// TIA Portal V18 export
// export: Created 2026-03-12T16:04:35.2784155Z, ExportSetting WithDefaults, DisplayName Totally Integrated Automation Portal, DisplayVersion V18 Update 5, DisplayName TIA Portal Openness, DisplayVersion V18 Update 5, DisplayName TIA Portal Version Control Interface, DisplayVersion V18, DisplayName SINAMICS Startdrive Advanced, DisplayVersion V18, DisplayName SINAMICS Startdrive G130, G150, S120, S150, SINAMICS MV, S210, DisplayVersion V18, DisplayName SINAMICS Startdrive G110M, G120, G120C, G120D, G120P, G115D, DisplayVersion V18, DisplayName STEP 7 Professional, DisplayVersion V18 Update 5, DisplayName STEP 7 Safety, DisplayVersion V18, DisplayName WinCC Professional, DisplayVersion V18 Update 5
FUNCTION_BLOCK "FB TOTALIZADOR"   // FB16, LAD
TITLE = Function Block TOTALIZADOR - Calculando os totalizadores dos macromedidores
{ S7_Optimized_Access := 'TRUE' }
VERSION : 0.1
// Network 1: Recebendo sinal de pulso
// Network 2: Primeira Soma (Incremento a cada 1 pulso)
// Network 3: Segunda Soma (Incremento a cada 1000 pulsos)
// Network 4: Resetando o totalizador
// stored: AutoNumber true, IsIECCheckEnabled false, IsRetainMemResEnabled false, MemoryReserve 100, SetENOAutomatically false, UDAEnableTagReadback false
   VAR_INPUT
      ENTRADA_SINAL : Bool;   // Entrada do sinal proveniente do hidrômetro/macromedidor
      RESET_TOT : Bool;   // Input de reset para zerar os blocos de incremento do totalizador
      MULTIPLICADOR_OUT : Real := 1.0;
      MANUTENCAO : Bool;
   END_VAR
   VAR_OUTPUT
      TOT_SAÍDA : UInt;   // Saída real do totalizador (m³)
   END_VAR
   VAR RETAIN
      PULSE1 : Bool;   // Pulso inicial para contar os sinais elétricos da entrada digital
      COUNT_PULSE1 : Bool;   // Contador de Pulsos 1
      PULSE2 : Bool;   // Rampa de subida para assegurar que o sinal da comparação anterior seja identificado como pulso pelo CLP
      COUNT_PULSE2 : Bool;   // Contador de pulsos 2
      SOMA1 : UInt;   // Bloco de incremento a cada pulso recebido na variável PULSE
      SOMA1_TOT_PREV : UInt;   // Variável que recebe a primeira soma
      SOMA2 : UInt;   // Variável que recebe o incremento de 1000 em 1000 e move ao TOT_SAÍDA Output para ser utilizado
      MULT_INC : UInt;   // Multiplicador da saída.
   END_VAR
   VAR_TEMP   // added for the SCL form of the ladder/FBD networks
      _w1 : Bool;
   END_VAR
BEGIN

REGION Network 1: Recebendo sinal de pulso
   // ENTRADA_SINAL: Input que recebe o sinal de pulso do equipamento
   // PULSE1: Rampa de subida para assegurar que o sinal recebido seja identificado como pulso pelo CLP
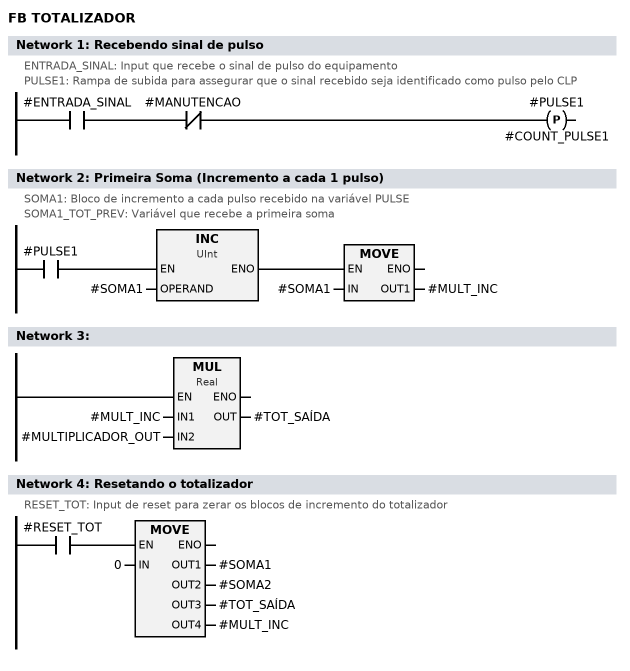
   #_w1 := #ENTRADA_SINAL AND NOT #MANUTENCAO;
   #PULSE1 := #_w1 AND NOT #COUNT_PULSE1;   // rising edge
   #COUNT_PULSE1 := #_w1;
END_REGION

REGION Network 2: Primeira Soma (Incremento a cada 1 pulso)
   // SOMA1: Bloco de incremento a cada pulso recebido na variável PULSE
   // SOMA1_TOT_PREV: Variável que recebe a primeira soma
   RUNG wire#powerrail
      Contact( #PULSE1 )
      { S7_Templates := "DestType := UInt" } Inc( #SOMA1 )
      Move(in := #SOMA1, out1 => #MULT_INC)
   END_RUNG
   // the same network as SCL:
   IF #PULSE1 THEN
       #SOMA1 := #SOMA1 + 1;
       #MULT_INC := #SOMA1;
   END_IF;
END_REGION

REGION Network 3
   RUNG wire#powerrail
      { S7_Templates := "SrcType := Real" } Mul(in1 := #MULT_INC, in2 := #MULTIPLICADOR_OUT, out => #TOT_SAÍDA)
   END_RUNG
   // the same network as SCL:
   #TOT_SAÍDA := #MULT_INC * #MULTIPLICADOR_OUT;
END_REGION

REGION Network 4: Resetando o totalizador
   // RESET_TOT: Input de reset para zerar os blocos de incremento do totalizador
   RUNG wire#powerrail
      Contact( #RESET_TOT )
      Move(in := 0, out1 => #SOMA1, out2 => #SOMA2, out3 => #TOT_SAÍDA, out4 => #MULT_INC)
   END_RUNG
   // the same network as SCL:
   IF #RESET_TOT THEN
       #SOMA1 := 0;
       #SOMA2 := 0;
       #TOT_SAÍDA := 0;
       #MULT_INC := 0;
   END_IF;
END_REGION
END_FUNCTION_BLOCK
